(* CoDeSys 2.3.9.41 project: testVariantAlgorithmToRegen.pro *)
(* Libraries: STANDARD.LIB 4.10.05 11:14:46, IECSFC.LIB 13.4.06 15:51:28, SYSLIBTIME.LIB 20.2.06 13:31:16, SYSTASKINFO.LIB 20.2.06 13:31:38, ANALYZATION.LIB 5.10.99 09:05:06, SYSLIBCALLBACK.LIB 20.2.06 13:31:08, Util.lib 18.5.10 15:14:28 *)

(* PLC configuration (modules and I/O channels)
PLC160 [Root] node -1, in %IB0 out %QB0 {MinCycleLength = 1; MaxCycleLength = 1000; MaxBackupTime = 6}
  Fast discrete inputs [I_SIMPLE_INPUT] node 0, in %IB0 out %QB0 {Filtrationtime = 10}
    AT %IX0.0 [BitInput] Discrete input 1
    AT %IX0.1 [BitInput] Discrete input 2
    AT %IX0.2 [BitInput] Discrete input 3
    AT %IX0.3 [BitInput] Discrete input 4
  Discrete inputs [ID130] node 1, in %IB1 out %QB1 {Filtrationtime_GeneralINP = 10; Visibility = No; PinCount = 12}
    AT %IB1.0 [ByteInput] 8 discrete inputs
    AT %IB1.1 [ByteInput] 4 discrete inputs
  Discrete outputs [ID131] node 2, in %IB2 out %QB2 {SafeValueByte = 0; SafeValueByteM = 0; Visibility = No; PinCount = 12}
    AT %QB2.0 [ByteOutput] 8 discrete outputs
    AT %QB2.1 [ByteOutput] 4 discrete outputs
  Fast analog inputs [ID125] node 3, in %IB3 out %QB3 {Flt_Comm = 50Hz 2Por}
    AT %IR3.0 [FloatInputP] AI #1 {AIN_TYPE = 4-20 mA; Peak_Filtr = 200; Flt_Ch = Off; TauRC = 10; MinFV = 0; MaxFV = 20000.0}
    AT %IR3.1 [FloatInputP] AI #2 {AIN_TYPE = 4-20 mA; Peak_Filtr = 200; Flt_Ch = Off; TauRC = 10; MinFV = 0; MaxFV = 20000.0}
    AT %IR3.2 [FloatInputP] AI #3 {AIN_TYPE = 4-20 mA; Peak_Filtr = 200; Flt_Ch = Off; TauRC = 10; MinFV = 0; MaxFV = 20000.0}
    AT %IR3.3 [FloatInputP] AI #4 {AIN_TYPE = 4-20 mA; Peak_Filtr = 200; Flt_Ch = Off; TauRC = 10; MinFV = 0; MaxFV = 20000.0}
    AT %IR3.4 [FloatInputP] AI #5 {AIN_TYPE = 4-20 mA; Peak_Filtr = 200; Flt_Ch = Off; TauRC = 10; MinFV = 0; MaxFV = 20000.0}
    AT %IR3.5 [FloatInputP] AI #6 {AIN_TYPE = 4-20 mA; Peak_Filtr = 200; Flt_Ch = Off; TauRC = 10; MinFV = 0; MaxFV = 20000.0}
    AT %IR3.6 [FloatInputP] AI #7 {AIN_TYPE = 4-20 mA; Peak_Filtr = 200; Flt_Ch = Off; TauRC = 10; MinFV = 0; MaxFV = 20000.0}
    AT %IR3.7 [FloatInputP] AI #8 {AIN_TYPE = 4-20 mA; Peak_Filtr = 200; Flt_Ch = Off; TauRC = 10; MinFV = 0; MaxFV = 20000.0}
    AT %IW3.8 [WordInput] AI read time (10ms)
  Analog outputs [ID126] node 4, in %IB4 out %QB4
    AT %QR4.0 [FloatOutputP] AO #1 {AOUT_TYPE = 4-20 mA; SafeValueREAL = 0.0}
    AT %QR4.1 [FloatOutputP] AO #2 {AOUT_TYPE = 4-20 mA; SafeValueREAL = 0.0}
    AT %QR4.2 [FloatOutputP] AO #3 {AOUT_TYPE = 4-20 mA; SafeValueREAL = 0.0}
    AT %QR4.3 [FloatOutputP] AO #4 {AOUT_TYPE = 4-20 mA; SafeValueREAL = 0.0}
  Special input [ID103] node 5, in %IB5 out %QB5 {Filtrationtime = 1000; PinCount = 1; WatchDogPeriod = 400; PollPeriod = 3000; Visibility = No}
    AT %IX5.0 [BitInput] Special input
  Special output [ID104] node 6, in %IB6 out %QB6 {Visibility = No; PinCount = 1}
    AT %QX6.0 [BitOutput] Special output
*)

(* POU PLC_PRG, CFC *)
PROGRAM PLC_PRG
VAR
	inputBlinker: BLINK;
	start: BOOL;
	sum: WORD;
	BlinkedAdder: F_TRIG;
	queueStarter: F_TRIG;
	queue: WORD;
	firstFilterRegen: BOOL;
	secondFilterRegen: BOOL;
	setToRegen: WORD;
	remainedToRegen: WORD;
	thirdFilterRegen: BOOL;
END_VAR
VAR (* helpers for the ST form of the networks *)
	_t43 : BOOL;
END_VAR
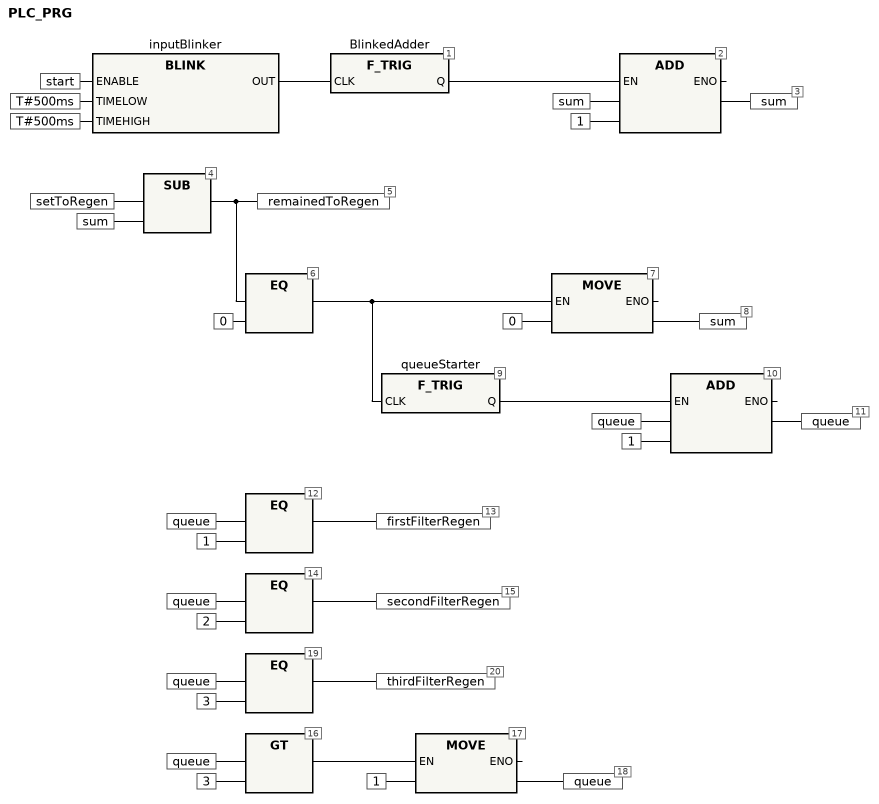
_CFC_ (* Continuous Function Chart, elements in execution order *)
#0 inputBlinker:BLINK(ENABLE: start, TIMELOW: T#500ms, TIMEHIGH: T#500ms)
#1 BlinkedAdder:F_TRIG(CLK: #0.OUT)
#2 ADD(EN: #1.Q, sum, 1)
#3 sum <= #2
#4 SUB(setToRegen, sum)
#5 remainedToRegen <= #4
#6 EQ(#4, 0)
#7 MOVE(EN: #6, 0)
#8 sum <= #7
#9 queueStarter:F_TRIG(CLK: #6)
#10 ADD(EN: #9.Q, queue, 1)
#11 queue <= #10
#12 EQ(queue, 1)
#13 firstFilterRegen <= #12
#14 EQ(queue, 2)
#15 secondFilterRegen <= #14
#16 GT(queue, 3)
#17 MOVE(EN: #16, 1)
#18 queue <= #17
#19 EQ(queue, 3)
#20 thirdFilterRegen <= #19
_END_CFC_
(* the same logic as Structured Text *)
inputBlinker(ENABLE := start, TIMELOW := T#500ms, TIMEHIGH := T#500ms);
BlinkedAdder(CLK := inputBlinker.OUT);
IF BlinkedAdder.Q THEN sum := sum + 1; END_IF;
remainedToRegen := setToRegen - sum;
_t43 := (setToRegen - sum) = 0;
IF _t43 THEN sum := 0; END_IF;
queueStarter(CLK := _t43);
IF queueStarter.Q THEN queue := queue + 1; END_IF;
firstFilterRegen := queue = 1;
secondFilterRegen := queue = 2;
IF queue > 3 THEN queue := 1; END_IF;
thirdFilterRegen := queue = 3;
END_PROGRAM
